FUNCTION_BLOCK FB_1_CargarBase_SFC
VAR_INPUT
	
	// Indicadores de sincronización
	Ack: BOOL := TRUE;
	Execute: BOOL;
	
	// Entradas
	PalePresencia AT %I*: BOOL;
	
END_VAR
VAR_OUTPUT
	
	// Indicadores de sincronización
	Ready: BOOL;	
	Done: BOOL;
	
	// Salidas
	CintaMotorActiva AT %Q*: BOOL;
	
END_VAR
VAR
END_VAR

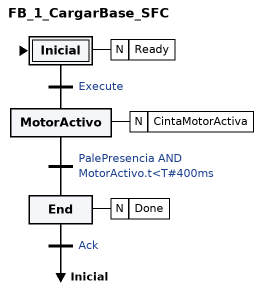
INITIAL_STEP Inicial:
    Ready(N);
END_STEP
TRANSITION FROM Inicial TO MotorActivo
    := Execute;
END_TRANSITION
STEP MotorActivo:
    CintaMotorActiva(N);
END_STEP
TRANSITION FROM MotorActivo TO End
    := PalePresencia AND MotorActivo.t<T#400ms;
END_TRANSITION
STEP End:
    Done(N);
END_STEP
TRANSITION FROM End TO Inicial
    := Ack;
END_TRANSITION

END_FUNCTION_BLOCK

(* stored: Version 1.1.0.1, ProductVersion 3.1.4024.12
   POU FB_1_CargarBase_SFC: Id {5fc7a0b4-0262-4f37-b54b-8dac773a28ac}, SpecialFunc None *)
